FUNCTION_BLOCK Q_ExecuteExtendedMacro_AUI (* Command Execute Extended Macro with AUI adapter ( Part 6 - F.62 ) *)
  (* Standard: ISO 11783-6; Description: Copyright (c) 2026 Meisterschulen am Ostbahnhof This program and the accompanying materials are made available under the terms of the Eclipse Public License 2.0 which is available at https://www.eclipse.org/legal/epl-2.0/ SPDX-License-Identifier: EPL-2.0 *)
  (* Version 1.0, 2026-09-11, Franz Höpfinger, Meisterschulen am Ostbahnhof, AUI adapter wrapper for Q_ExecuteExtendedMacro *)
  PACKAGE isobus::UT::Q;
  (* Documentation:
  Command Execute Extended Macro with AUI adapter ( Part 6 - F.62 )
   This FB is an AUI adapter wrapper around Q_ExecuteExtendedMacro.
  *)
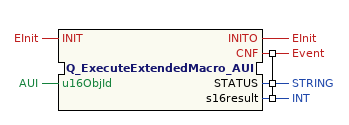
  EVENT_INPUT
    INIT : EInit; (* Service Initialization *)
  END_EVENT
  EVENT_OUTPUT
    INITO : EInit; (* Initialization Confirm *)
    CNF WITH STATUS, s16result; (* Confirmation of Requested Service *)
  END_EVENT
  VAR_OUTPUT
    STATUS : STRING; (* Service Status *)
    s16result : INT; (* retval see description *)
  END_VAR
  SOCKETS
    u16ObjId : adapter::types::unidirectional::AUI; (* Object ID of Macro object (range 1 - 999) *)
  END_SOCKETS
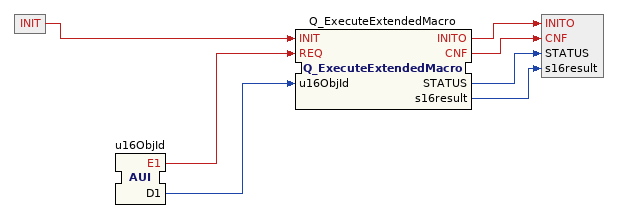
  FBS
    Q_ExecuteExtendedMacro : isobus::UT::Q::Q_ExecuteExtendedMacro;
  END_FBS
  EVENT_CONNECTIONS
    INIT TO Q_ExecuteExtendedMacro.INIT;
    Q_ExecuteExtendedMacro.INITO TO INITO;
    Q_ExecuteExtendedMacro.CNF TO CNF;
    u16ObjId.E1 TO Q_ExecuteExtendedMacro.REQ;
  END_CONNECTIONS
  DATA_CONNECTIONS
    Q_ExecuteExtendedMacro.STATUS TO STATUS;
    u16ObjId.D1 TO Q_ExecuteExtendedMacro.u16ObjId;
    Q_ExecuteExtendedMacro.s16result TO s16result;
  END_CONNECTIONS
END_FUNCTION_BLOCK
